(* PLC project PLCOpen_Leer.project, CODESYS CODESYS V3.5 SP7 Patch 2 *)
(* stored: creationDateTime 2018-07-08T13:58:46.9898301, modificationDateTime 2018-07-08T13:57:47.963454 *)

PROGRAM hhh
  VAR
    F1 : F_trig;
  END_VAR

		  	  
		  		;
		  		
		  	  
		  	
END_PROGRAM
